FUNCTION_BLOCK FB_InternalPowerSupply_IO

VAR_INPUT 
	b_DCPsuEnable		AT %Q* : BOOL := FALSE;
	b_ACPsuEnable		AT %Q* : BOOL := TRUE;
END_VAR

VAR_OUTPUT
	DCPSU_OK 			AT %I*: BOOL;
	ACPSU_OK 			AT %I*: BOOL;
	GridFuseOK 			AT %I*: BOOL;
END_VAR

END_FUNCTION_BLOCK

(* stored: Version 1.1.0.1, ProductVersion 3.1.4026.18
   POU FB_InternalPowerSupply_IO: Id {14a37718-20e2-4b4a-9114-4d8672574bf3}, SpecialFunc None *)
